PROGRAM MAIN
VAR
	bLED1 AT %Q*: BOOL;
	fbTON: TON := (PT := TIME#100MS);
END_VAR

fbTON(IN:= not(fbTON.Q), Q=>bLED1);

END_PROGRAM

(* stored: Version 1.1.0.1, ProductVersion 3.1.4024.12
   POU MAIN: Id {29ad1771-f66d-4994-99ae-8c562b978f26}, SpecialFunc None *)
